// TIA Portal V18 export
// export: Created 2026-03-12T16:04:32.0334217Z, ExportSetting WithDefaults, DisplayName Totally Integrated Automation Portal, DisplayVersion V18 Update 5, DisplayName TIA Portal Openness, DisplayVersion V18 Update 5, DisplayName TIA Portal Version Control Interface, DisplayVersion V18, DisplayName SINAMICS Startdrive Advanced, DisplayVersion V18, DisplayName SINAMICS Startdrive G130, G150, S120, S150, SINAMICS MV, S210, DisplayVersion V18, DisplayName SINAMICS Startdrive G110M, G120, G120C, G120D, G120P, G115D, DisplayVersion V18, DisplayName STEP 7 Professional, DisplayVersion V18 Update 5, DisplayName STEP 7 Safety, DisplayVersion V18, DisplayName WinCC Professional, DisplayVersion V18 Update 5
DATA_BLOCK "FB INTERTRAVAMENTO_PAINEL_CA-02"   // DB598
VERSION : 0.1
// stored: AutoNumber true, DBAccessibleFromOPCUA true, DBAccessibleFromWebserver true, InstanceOfName FB INTERTRAVAMENTO_PAINEL, InstanceOfType FB
"FB INTERTRAVAMENTO_PAINEL"
   // VAR_INPUT
   //    INPUT_BT_EMERGENCIA : Bool;
   //    INPUT_DISJUNTOR : Bool;
   //    INPUT_FONTE1 : Bool;
   //    INPUT_FONTE2 : Bool;
   //    INPUT_RELE_FALTA : Bool;
   //    INPUT_CONDICAO : Bool;
   //    INPUT_TESTE : Bool;
   // END_VAR
   // VAR_OUTPUT
   //    OUTPUT_PAINEL_OK : Bool;
   // END_VAR
BEGIN
END_DATA_BLOCK
